// TIA Portal V17 export
// export: Created 2023-02-26T22:57:58.6071469Z, ExportSetting WithDefaults, DisplayName Totally Integrated Automation Portal, DisplayVersion V17, DisplayName TIA Portal Openness, DisplayVersion V17, DisplayName TIA Portal Version Control Interface, DisplayVersion V17, DisplayName TIA Portal Test Suite Advanced, DisplayVersion V17, DisplayName STEP 7 Professional, DisplayVersion V17, DisplayName SIMATIC Energy Suite, DisplayVersion V17, DisplayName STEP 7 Safety, DisplayVersion V17, DisplayName WinCC Professional, DisplayVersion V17
FUNCTION "LOG_CountModes" : Void   // FC19, LAD
{ S7_Optimized_Access := 'TRUE' }
VERSION : 0.1
// stored: AutoNumber true, IsIECCheckEnabled false, SetENOAutomatically false, UDAEnableTagReadback false
BEGIN

REGION Network 1: Call: CountMode - Auto
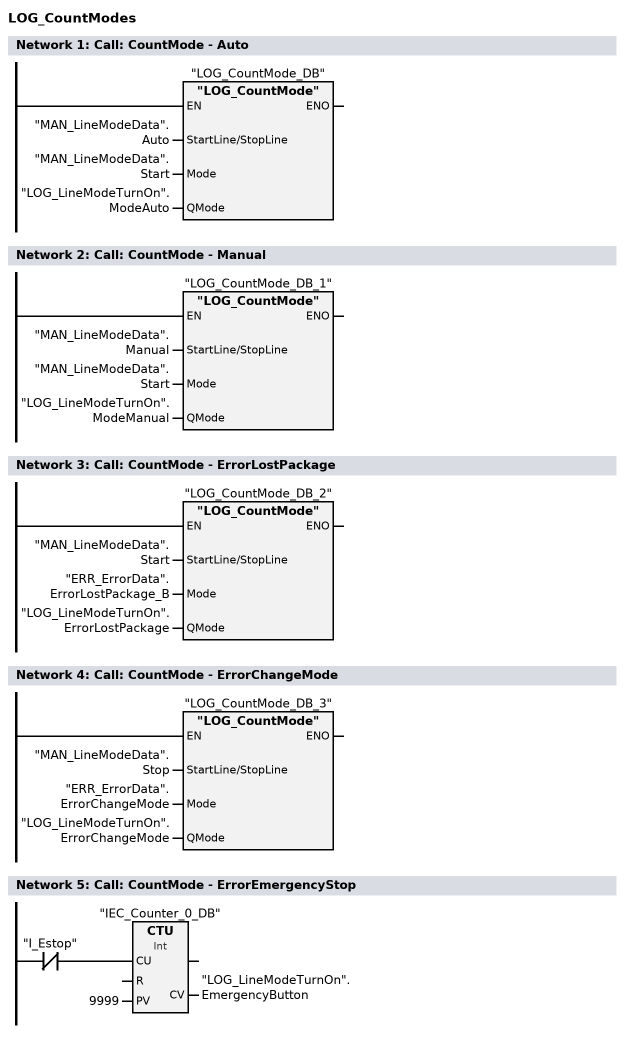
   RUNG wire#powerrail
      "LOG_CountMode_DB"("StartLine/StopLine" := "MAN_LineModeData".Auto, Mode := "MAN_LineModeData".Start, QMode := "LOG_LineModeTurnOn".ModeAuto)
   END_RUNG
   // the same network as SCL:
   "LOG_CountMode_DB"("StartLine/StopLine" := "MAN_LineModeData".Auto,   // "LOG_CountMode"
                      Mode := "MAN_LineModeData".Start,
                      QMode := "LOG_LineModeTurnOn".ModeAuto);
END_REGION

REGION Network 2: Call: CountMode - Manual
   RUNG wire#powerrail
      "LOG_CountMode_DB_1"("StartLine/StopLine" := "MAN_LineModeData".Manual, Mode := "MAN_LineModeData".Start, QMode := "LOG_LineModeTurnOn".ModeManual)
   END_RUNG
   // the same network as SCL:
   "LOG_CountMode_DB_1"("StartLine/StopLine" := "MAN_LineModeData".Manual,   // "LOG_CountMode"
                        Mode := "MAN_LineModeData".Start,
                        QMode := "LOG_LineModeTurnOn".ModeManual);
END_REGION

REGION Network 3: Call: CountMode - ErrorLostPackage
   RUNG wire#powerrail
      "LOG_CountMode_DB_2"("StartLine/StopLine" := "MAN_LineModeData".Start, Mode := "ERR_ErrorData".ErrorLostPackage_B, QMode := "LOG_LineModeTurnOn".ErrorLostPackage)
   END_RUNG
   // the same network as SCL:
   "LOG_CountMode_DB_2"("StartLine/StopLine" := "MAN_LineModeData".Start,   // "LOG_CountMode"
                        Mode := "ERR_ErrorData".ErrorLostPackage_B,
                        QMode := "LOG_LineModeTurnOn".ErrorLostPackage);
END_REGION

REGION Network 4: Call: CountMode - ErrorChangeMode
   RUNG wire#powerrail
      "LOG_CountMode_DB_3"("StartLine/StopLine" := "MAN_LineModeData".Stop, Mode := "ERR_ErrorData".ErrorChangeMode, QMode := "LOG_LineModeTurnOn".ErrorChangeMode)
   END_RUNG
   // the same network as SCL:
   "LOG_CountMode_DB_3"("StartLine/StopLine" := "MAN_LineModeData".Stop,   // "LOG_CountMode"
                        Mode := "ERR_ErrorData".ErrorChangeMode,
                        QMode := "LOG_LineModeTurnOn".ErrorChangeMode);
END_REGION

REGION Network 5: Call: CountMode - ErrorEmergencyStop
   RUNG wire#powerrail
      I_Contact( "I_Estop" )
      { S7_Templates := "value_type := Int" } "IEC_Counter_0_DB".CTU(r :=, pv := 9999, cv => "LOG_LineModeTurnOn".EmergencyButton)
   END_RUNG
   // the same network as SCL:
   "IEC_Counter_0_DB".CTU(CU := NOT "I_Estop", PV := 9999, CV => "LOG_LineModeTurnOn".EmergencyButton);
END_REGION
END_FUNCTION
